Staubli VAL3: SIMPLE_MSG.pgx

program SIMPLE_MSG(num x_nLength, num x_nMsgType)
  local num l_nStatus
  local num l_nBytesToGet
  local num i
  local num j
  local num k
  local num l_nRespBuffer[152]
  local joint l_jJoint
  local mdesc l_mMdesc
begin
  // This TASK specialises in receiving ros simple messages
  // thus it validates prefix and the header and then accepts
  // the bytes from the body
  // payload length in bytes minus header size (12 bytes)
  l_nBytesToGet=x_nLength-12
  resize(nInputBuffer,1,l_nBytesToGet)
  resize(nMessageBuffer,1,l_nBytesToGet/4)
  resize(nMessageBuffer,2,4)
  while (bInputBuffering)
    l_nStatus=0
    // prefix
    call consume(l_nStatus,x_nLength)
    // header
    call consume(l_nStatus,x_nMsgType)
    call consume(l_nStatus,msgSpec:commType.nRequest)
    call consumeAny(l_nStatus)
    if l_nStatus<0
      if l_nStatus==-2
        putln("Timeout.")
      else
        putln("Bad request header/prefix.")
      endIf
    else
      // get the body
      j=0
      k=0
      while j<l_nBytesToGet/4
        l_nStatus=sioGet(siConn,nInputBuffer)
        if l_nStatus>0
          for i=0 to l_nStatus-1
            nMessageBuffer[j,k]=nInputBuffer[i]
            k=k+1
            if k>3
              k=0
              j=j+1
            endIf
          endFor
        endIf
      endWhile
      // decode the body
      call trajMsg:decode(l_nStatus,nMessageBuffer)
      delay(0)
      // modify the header for acknowledge message
      trajMsg:header.nCommType=msgSpec:commType.nResponse
      if l_nStatus<0
        trajMsg:header.nReplyCode=msgSpec:replyType.nFailure
        putln("Failed to decode the body of the message.")
      else
        trajMsg:header.nReplyCode=msgSpec:replyType.nSuccess
      endIf
      // encode the acknowledge message
      call trajMsg:encode(l_nStatus,l_nRespBuffer)
      if l_nStatus<0
        putln("Failed to encode the acknowledge message.")
        trajMsg:header.nReplyCode=msgSpec:replyType.nFailure
      endIf
      // send the acknowledge message
      l_nStatus=sioSet(soConn,l_nRespBuffer)
      if l_nStatus<0
        putln("Failed to send acknowledge response: "+toString("",l_nStatus))
      else
        // convert the message to joint & motion descirptor
        call trajMsg:convert(l_jJoint,l_mMdesc)
        // print the joint values
        put(toString("5",l_jJoint.j1)+","+toString("5",l_jJoint.j2)+","+toString("5",l_jJoint.j3))
        putln(","+toString("5",l_jJoint.j4)+","+toString("5",l_jJoint.j5)+","+toString("5",l_jJoint.j6))
        // apply the point to flange and add it to the motion queue
        movej(l_jJoint,flange,l_mMdesc)
      endIf
    endIf
  endWhile
end
